// TIA Portal V20 export
TYPE "LConSMC_typeKpAdaption"
// Ein-/Ausgänge der Drehzahlregler Kp-Adaption / In-/Outputs of the speed controller Kp-Adaption
// stored: Access Published
   STRUCT
      in { S7_SetPoint := 'True'} : "LConSMC_typeKpAdaptionInput";   // Eingänge des Bausteins KpAdaption / Inputs for FB KpAdaption
      out { S7_SetPoint := 'True'} : "LConSMC_typeKpAdaptionOutput";   // Ausgänge des Bausteins KpAdaption / Outputs for FB KpAdaption
   END_STRUCT;
END_TYPE
